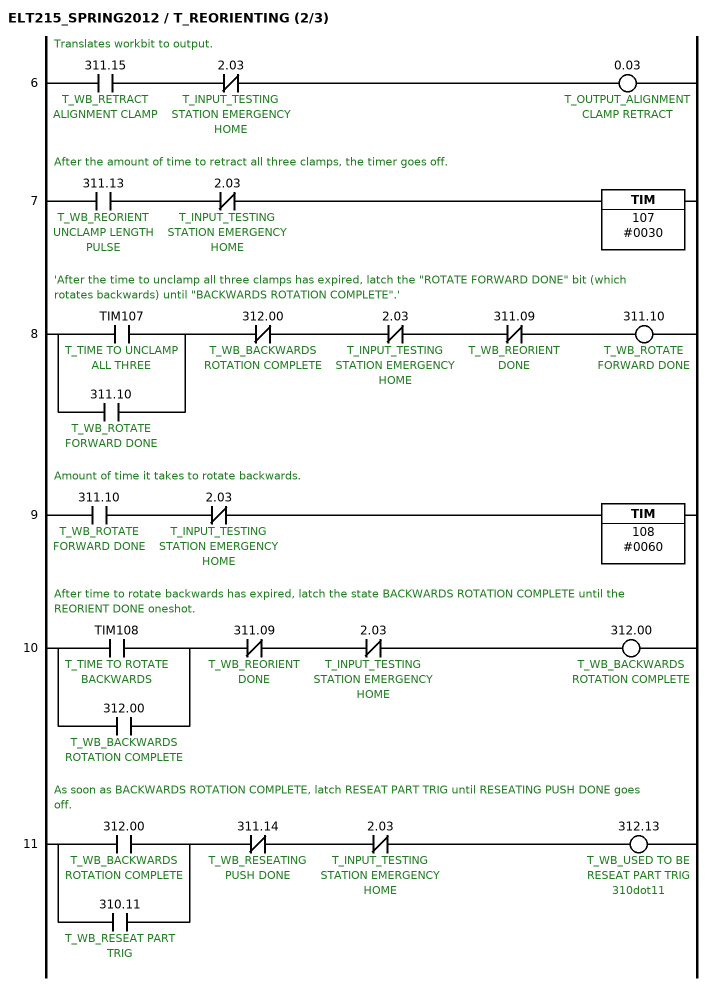
; [picture p24: ELT215_SPRING2012 / T_REORIENTING, rungs 6-11]
; rung 6: Translates workbit to output.
LD 311.15  ; T_WB_RETRACT ALIGNMENT CLAMP
ANDNOT 2.03  ; T_INPUT_TESTING STATION EMERGENCY HOME
OUT 0.03  ; T_OUTPUT_ALIGNMENT CLAMP RETRACT
; rung 7: After the amount of time to retract all three clamps, the timer goes off.
LD 311.13  ; T_WB_REORIENT UNCLAMP LENGTH PULSE
ANDNOT 2.03  ; T_INPUT_TESTING STATION EMERGENCY HOME
TIM 107 #0030
; rung 8: 'After the time to unclamp all three clamps has expired, latch the "ROTATE FORWARD DONE" bit (which rotates backwards) until "BACKWARDS ROTATION COMPLETE".'
LD TIM107  ; T_TIME TO UNCLAMP ALL THREE
OR 311.10  ; T_WB_ROTATE FORWARD DONE
ANDNOT 312.00  ; T_WB_BACKWARDS ROTATION COMPLETE
ANDNOT 2.03  ; T_INPUT_TESTING STATION EMERGENCY HOME
ANDNOT 311.09  ; T_WB_REORIENT DONE
OUT 311.10  ; T_WB_ROTATE FORWARD DONE
; rung 9: Amount of time it takes to rotate backwards.
LD 311.10  ; T_WB_ROTATE FORWARD DONE
ANDNOT 2.03  ; T_INPUT_TESTING STATION EMERGENCY HOME
TIM 108 #0060
; rung 10: After time to rotate backwards has expired, latch the state BACKWARDS ROTATION COMPLETE until the REORIENT DONE oneshot.
LD TIM108  ; T_TIME TO ROTATE BACKWARDS
OR 312.00  ; T_WB_BACKWARDS ROTATION COMPLETE
ANDNOT 311.09  ; T_WB_REORIENT DONE
ANDNOT 2.03  ; T_INPUT_TESTING STATION EMERGENCY HOME
OUT 312.00  ; T_WB_BACKWARDS ROTATION COMPLETE
; rung 11: As soon as BACKWARDS ROTATION COMPLETE, latch RESEAT PART TRIG until RESEATING PUSH DONE goes off.
LD 312.00  ; T_WB_BACKWARDS ROTATION COMPLETE
OR 310.11  ; T_WB_RESEAT PART TRIG
ANDNOT 311.14  ; T_WB_RESEATING PUSH DONE
ANDNOT 2.03  ; T_INPUT_TESTING STATION EMERGENCY HOME
OUT 312.13  ; T_WB_USED TO BE RESEAT PART TRIG 310dot11

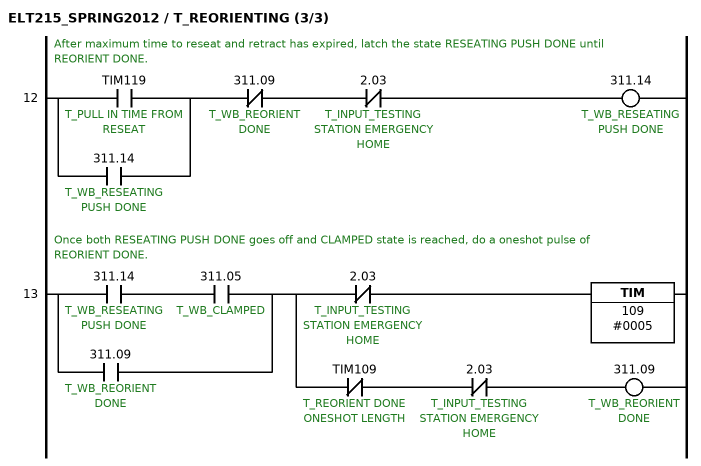
; rung 12: After maximum time to reseat and retract has expired, latch the state RESEATING PUSH DONE until REORIENT DONE.
LD TIM119  ; T_PULL IN TIME FROM RESEAT
OR 311.14  ; T_WB_RESEATING PUSH DONE
ANDNOT 311.09  ; T_WB_REORIENT DONE
ANDNOT 2.03  ; T_INPUT_TESTING STATION EMERGENCY HOME
OUT 311.14  ; T_WB_RESEATING PUSH DONE
; rung 13: Once both RESEATING PUSH DONE goes off and CLAMPED state is reached, do a oneshot pulse of REORIENT DONE.
LD 311.14  ; T_WB_RESEATING PUSH DONE
AND 311.05  ; T_WB_CLAMPED
OR 311.09  ; T_WB_REORIENT DONE
OUT TR0
ANDNOT 2.03  ; T_INPUT_TESTING STATION EMERGENCY HOME
TIM 109 #0005
LD TR0
ANDNOT TIM109  ; T_REORIENT DONE ONESHOT LENGTH
ANDNOT 2.03  ; T_INPUT_TESTING STATION EMERGENCY HOME
OUT 311.09  ; T_WB_REORIENT DONE

### Section T_HOLD_FOR_TESTING
; Ladder logic that can accept a tier 2 request to hold the part for testing (identified as being properly oriented) and can perform the actions to hold the piece, run the test sequence, and then eject the piece from the system.

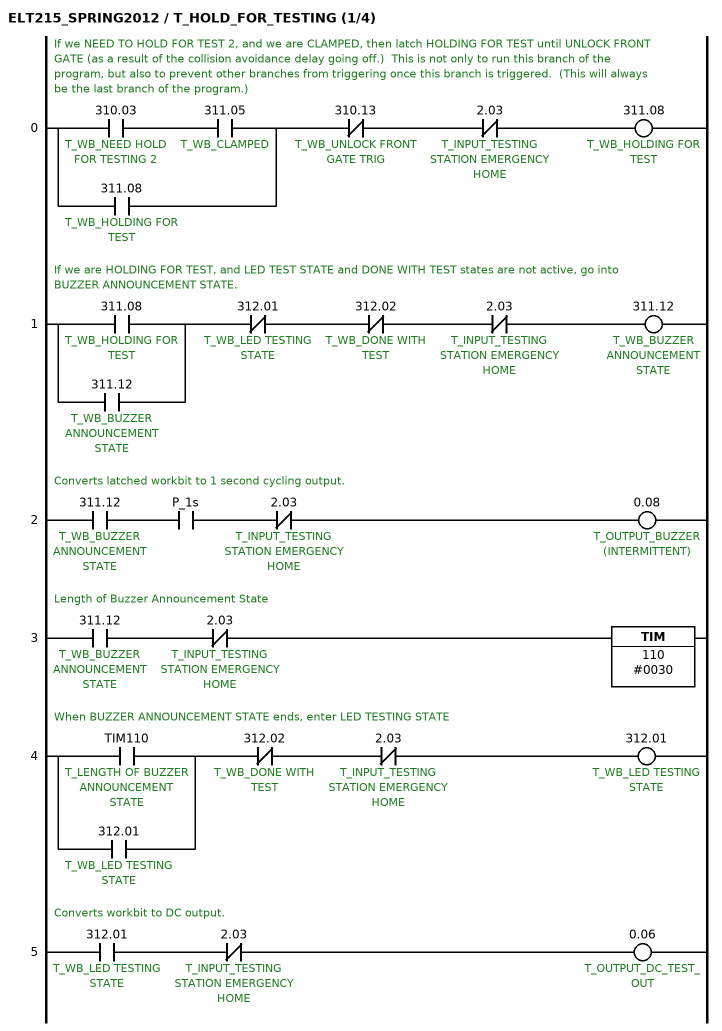
; rung 0: If we NEED TO HOLD FOR TEST 2, and we are CLAMPED, then latch HOLDING FOR TEST until UNLOCK FRONT GATE (as a result of the collision avoidance delay going off.)  This is not only to run this branch of the program, but also to prevent other branches from triggering once this branch is triggered.  (This will always be the last branch of the program.)
LD 310.03  ; T_WB_NEED HOLD FOR TESTING 2
AND 311.05  ; T_WB_CLAMPED
OR 311.08  ; T_WB_HOLDING FOR TEST
ANDNOT 310.13  ; T_WB_UNLOCK FRONT GATE TRIG
ANDNOT 2.03  ; T_INPUT_TESTING STATION EMERGENCY HOME
OUT 311.08  ; T_WB_HOLDING FOR TEST
; rung 1: If we are HOLDING FOR TEST, and LED TEST STATE and DONE WITH TEST states are not active, go into BUZZER ANNOUNCEMENT STATE.
LD 311.08  ; T_WB_HOLDING FOR TEST
OR 311.12  ; T_WB_BUZZER ANNOUNCEMENT STATE
ANDNOT 312.01  ; T_WB_LED TESTING STATE
ANDNOT 312.02  ; T_WB_DONE WITH TEST
ANDNOT 2.03  ; T_INPUT_TESTING STATION EMERGENCY HOME
OUT 311.12  ; T_WB_BUZZER ANNOUNCEMENT STATE
; rung 2: Converts latched workbit to 1 second cycling output.
LD 311.12  ; T_WB_BUZZER ANNOUNCEMENT STATE
AND P_1s
ANDNOT 2.03  ; T_INPUT_TESTING STATION EMERGENCY HOME
OUT 0.08  ; T_OUTPUT_BUZZER (INTERMITTENT)
; rung 3: Length of Buzzer Announcement State
LD 311.12  ; T_WB_BUZZER ANNOUNCEMENT STATE
ANDNOT 2.03  ; T_INPUT_TESTING STATION EMERGENCY HOME
TIM 110 #0030
; rung 4: When BUZZER ANNOUNCEMENT STATE ends, enter LED TESTING STATE
LD TIM110  ; T_LENGTH OF BUZZER ANNOUNCEMENT STATE
OR 312.01  ; T_WB_LED TESTING STATE
ANDNOT 312.02  ; T_WB_DONE WITH TEST
ANDNOT 2.03  ; T_INPUT_TESTING STATION EMERGENCY HOME
OUT 312.01  ; T_WB_LED TESTING STATE
; rung 5: Converts workbit to DC output.
LD 312.01  ; T_WB_LED TESTING STATE
ANDNOT 2.03  ; T_INPUT_TESTING STATION EMERGENCY HOME
OUT 0.06  ; T_OUTPUT_DC_TEST_OUT

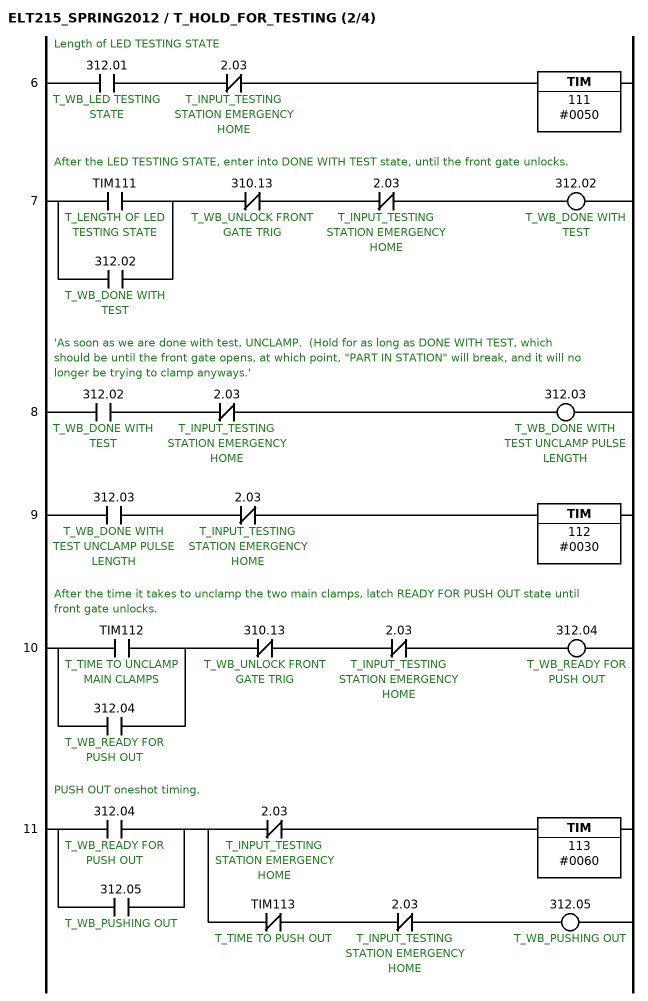
; rung 6: Length of LED TESTING STATE
LD 312.01  ; T_WB_LED TESTING STATE
ANDNOT 2.03  ; T_INPUT_TESTING STATION EMERGENCY HOME
TIM 111 #0050
; rung 7: After the LED TESTING STATE, enter into DONE WITH TEST state, until the front gate unlocks.
LD TIM111  ; T_LENGTH OF LED TESTING STATE
OR 312.02  ; T_WB_DONE WITH TEST
ANDNOT 310.13  ; T_WB_UNLOCK FRONT GATE TRIG
ANDNOT 2.03  ; T_INPUT_TESTING STATION EMERGENCY HOME
OUT 312.02  ; T_WB_DONE WITH TEST
; rung 8: 'As soon as we are done with test, UNCLAMP.  (Hold for as long as DONE WITH TEST, which should be until the front gate opens, at which point, "PART IN STATION" will break, and it will no longer be trying to clamp anyways.'
LD 312.02  ; T_WB_DONE WITH TEST
ANDNOT 2.03  ; T_INPUT_TESTING STATION EMERGENCY HOME
OUT 312.03  ; T_WB_DONE WITH TEST UNCLAMP PULSE LENGTH
; rung 9
LD 312.03  ; T_WB_DONE WITH TEST UNCLAMP PULSE LENGTH
ANDNOT 2.03  ; T_INPUT_TESTING STATION EMERGENCY HOME
TIM 112 #0030
; rung 10: After the time it takes to unclamp the two main clamps, latch READY FOR PUSH OUT state until front gate unlocks.
LD TIM112  ; T_TIME TO UNCLAMP MAIN CLAMPS
OR 312.04  ; T_WB_READY FOR PUSH OUT
ANDNOT 310.13  ; T_WB_UNLOCK FRONT GATE TRIG
ANDNOT 2.03  ; T_INPUT_TESTING STATION EMERGENCY HOME
OUT 312.04  ; T_WB_READY FOR PUSH OUT
; rung 11: PUSH OUT oneshot timing.
LD 312.04  ; T_WB_READY FOR PUSH OUT
OR 312.05  ; T_WB_PUSHING OUT
OUT TR0
ANDNOT 2.03  ; T_INPUT_TESTING STATION EMERGENCY HOME
TIM 113 #0060
LD TR0
ANDNOT TIM113  ; T_TIME TO PUSH OUT
ANDNOT 2.03  ; T_INPUT_TESTING STATION EMERGENCY HOME
OUT 312.05  ; T_WB_PUSHING OUT

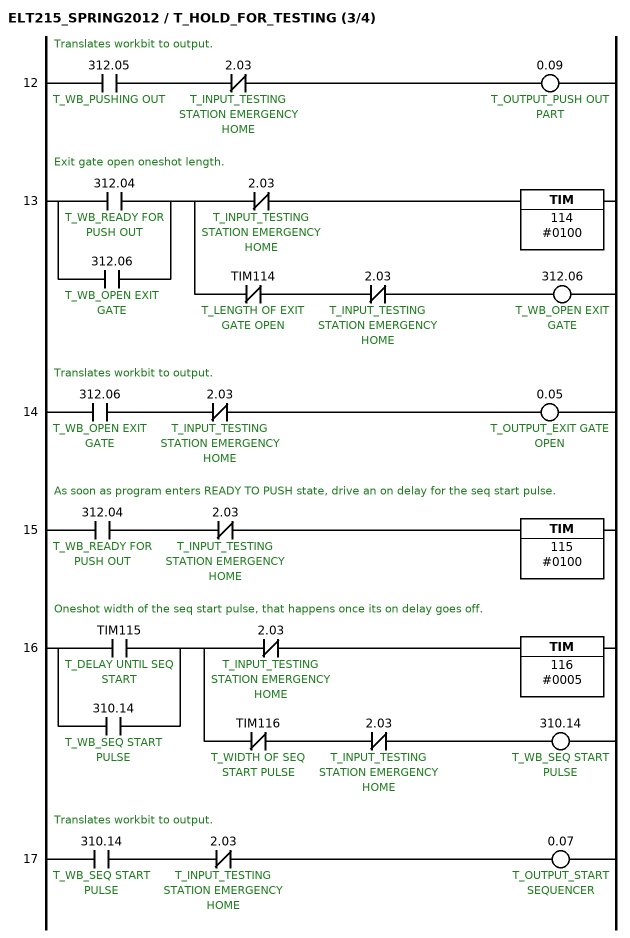
; rung 12: Translates workbit to output.
LD 312.05  ; T_WB_PUSHING OUT
ANDNOT 2.03  ; T_INPUT_TESTING STATION EMERGENCY HOME
OUT 0.09  ; T_OUTPUT_PUSH OUT PART
; rung 13: Exit gate open oneshot length.
LD 312.04  ; T_WB_READY FOR PUSH OUT
OR 312.06  ; T_WB_OPEN EXIT GATE
OUT TR0
ANDNOT 2.03  ; T_INPUT_TESTING STATION EMERGENCY HOME
TIM 114 #0100
LD TR0
ANDNOT TIM114  ; T_LENGTH OF EXIT GATE OPEN
ANDNOT 2.03  ; T_INPUT_TESTING STATION EMERGENCY HOME
OUT 312.06  ; T_WB_OPEN EXIT GATE
; rung 14: Translates workbit to output.
LD 312.06  ; T_WB_OPEN EXIT GATE
ANDNOT 2.03  ; T_INPUT_TESTING STATION EMERGENCY HOME
OUT 0.05  ; T_OUTPUT_EXIT GATE OPEN
; rung 15: As soon as program enters READY TO PUSH state, drive an on delay for the seq start pulse.
LD 312.04  ; T_WB_READY FOR PUSH OUT
ANDNOT 2.03  ; T_INPUT_TESTING STATION EMERGENCY HOME
TIM 115 #0100
; rung 16: Oneshot width of the seq start pulse, that happens once its on delay goes off.
LD TIM115  ; T_DELAY UNTIL SEQ START
OR 310.14  ; T_WB_SEQ START PULSE
OUT TR0
ANDNOT 2.03  ; T_INPUT_TESTING STATION EMERGENCY HOME
TIM 116 #0005
LD TR0
ANDNOT TIM116  ; T_WIDTH OF SEQ START PULSE
ANDNOT 2.03  ; T_INPUT_TESTING STATION EMERGENCY HOME
OUT 310.14  ; T_WB_SEQ START PULSE
; rung 17: Translates workbit to output.
LD 310.14  ; T_WB_SEQ START PULSE
ANDNOT 2.03  ; T_INPUT_TESTING STATION EMERGENCY HOME
OUT 0.07  ; T_OUTPUT_START SEQUENCER

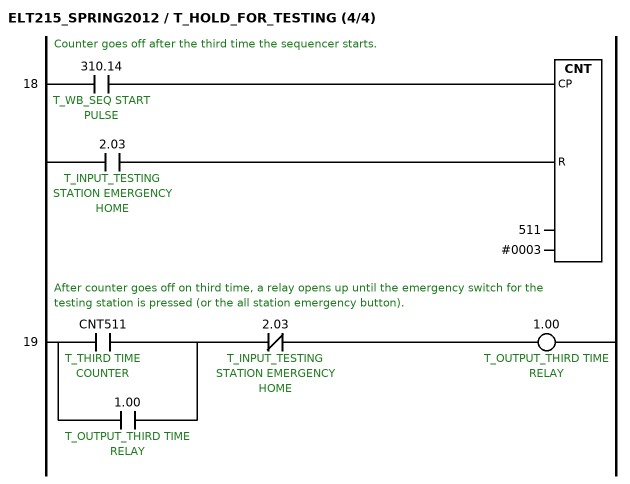
; rung 18: Counter goes off after the third time the sequencer starts.
LD 310.14  ; T_WB_SEQ START PULSE
LD 2.03  ; T_INPUT_TESTING STATION EMERGENCY HOME
CNT 511 #0003
; rung 19: After counter goes off on third time, a relay opens up until the emergency switch for the testing station is pressed (or the all station emergency button).
LD CNT511  ; T_THIRD TIME COUNTER
OR 1.00  ; T_OUTPUT_THIRD TIME RELAY
ANDNOT 2.03  ; T_INPUT_TESTING STATION EMERGENCY HOME
OUT 1.00  ; T_OUTPUT_THIRD TIME RELAY

### Section T_SYSTEM_RESET_AND_ABORT
; Ladder logic that defines the two different ways the program can end and reset.  A. Through an abort command  B. Through a SEQ START pulse, which will then get delayed to avoid a possible collision if the next part comes in properly oriented.

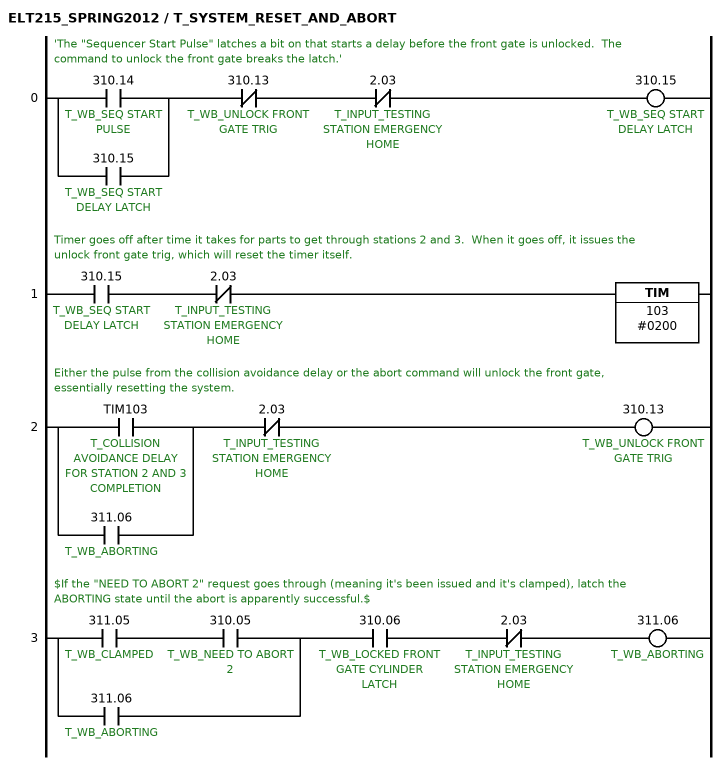
; rung 0: 'The "Sequencer Start Pulse" latches a bit on that starts a delay before the front gate is unlocked.  The command to unlock the front gate breaks the latch.'
LD 310.14  ; T_WB_SEQ START PULSE
OR 310.15  ; T_WB_SEQ START DELAY LATCH
ANDNOT 310.13  ; T_WB_UNLOCK FRONT GATE TRIG
ANDNOT 2.03  ; T_INPUT_TESTING STATION EMERGENCY HOME
OUT 310.15  ; T_WB_SEQ START DELAY LATCH
; rung 1: Timer goes off after time it takes for parts to get through stations 2 and 3.  When it goes off, it issues the unlock front gate trig, which will reset the timer itself.
LD 310.15  ; T_WB_SEQ START DELAY LATCH
ANDNOT 2.03  ; T_INPUT_TESTING STATION EMERGENCY HOME
TIM 103 #0200
; rung 2: Either the pulse from the collision avoidance delay or the abort command will unlock the front gate, essentially resetting the system.
LD TIM103  ; T_COLLISION AVOIDANCE DELAY FOR STATION 2 AND 3 COMPLETION
OR 311.06  ; T_WB_ABORTING
ANDNOT 2.03  ; T_INPUT_TESTING STATION EMERGENCY HOME
OUT 310.13  ; T_WB_UNLOCK FRONT GATE TRIG
; rung 3: $If the "NEED TO ABORT 2" request goes through (meaning it's been issued and it's clamped), latch the ABORTING state until the abort is apparently successful.$
LD 311.05  ; T_WB_CLAMPED
AND 310.05  ; T_WB_NEED TO ABORT 2
OR 311.06  ; T_WB_ABORTING
AND 310.06  ; T_WB_LOCKED FRONT GATE CYLINDER LATCH
ANDNOT 2.03  ; T_INPUT_TESTING STATION EMERGENCY HOME
OUT 311.06  ; T_WB_ABORTING

### Section T_OBSERVATION_ONLY

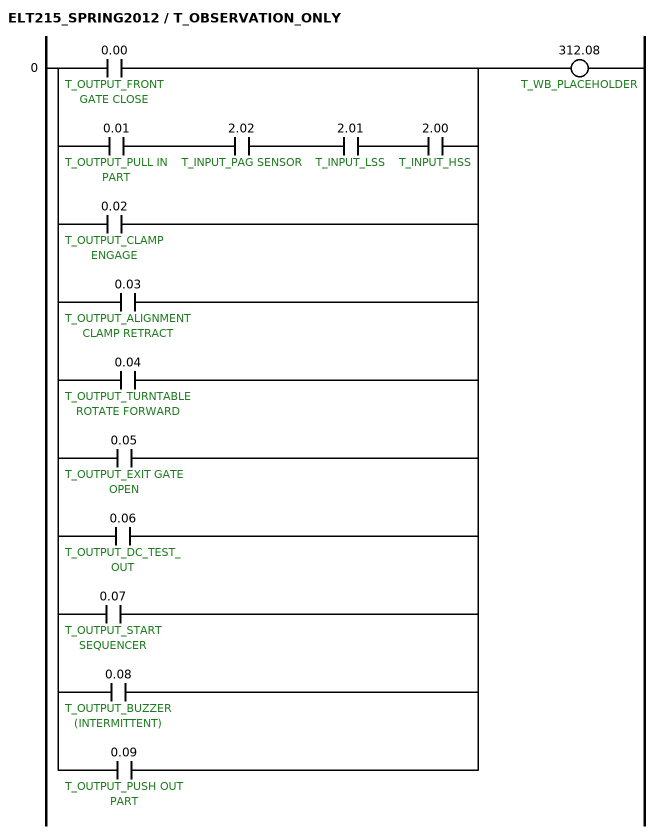
; rung 0
LD 0.00  ; T_OUTPUT_FRONT GATE CLOSE
LD 0.01  ; T_OUTPUT_PULL IN PART
AND 2.02  ; T_INPUT_PAG SENSOR
AND 2.01  ; T_INPUT_LSS
AND 2.00  ; T_INPUT_HSS
ORLD
LD 0.02  ; T_OUTPUT_CLAMP ENGAGE
OR 0.03  ; T_OUTPUT_ALIGNMENT CLAMP RETRACT
OR 0.04  ; T_OUTPUT_TURNTABLE ROTATE FORWARD
OR 0.05  ; T_OUTPUT_EXIT GATE OPEN
OR 0.06  ; T_OUTPUT_DC_TEST_OUT
OR 0.07  ; T_OUTPUT_START SEQUENCER
OR 0.08  ; T_OUTPUT_BUZZER (INTERMITTENT)
OR 0.09  ; T_OUTPUT_PUSH OUT PART
ORLD
OUT 312.08  ; T_WB_PLACEHOLDER

### Section F_FEEDER_SEQUENCE_TIME
; 'Offset from T=0, contains timings for the ejection of each part, as well as the "SEQUENCE OVER" point.  For example, if parts are supposed to come out at ten second intervals, part 1 would be released at 0, part 2 at 10, part 3 at 20, etc.'

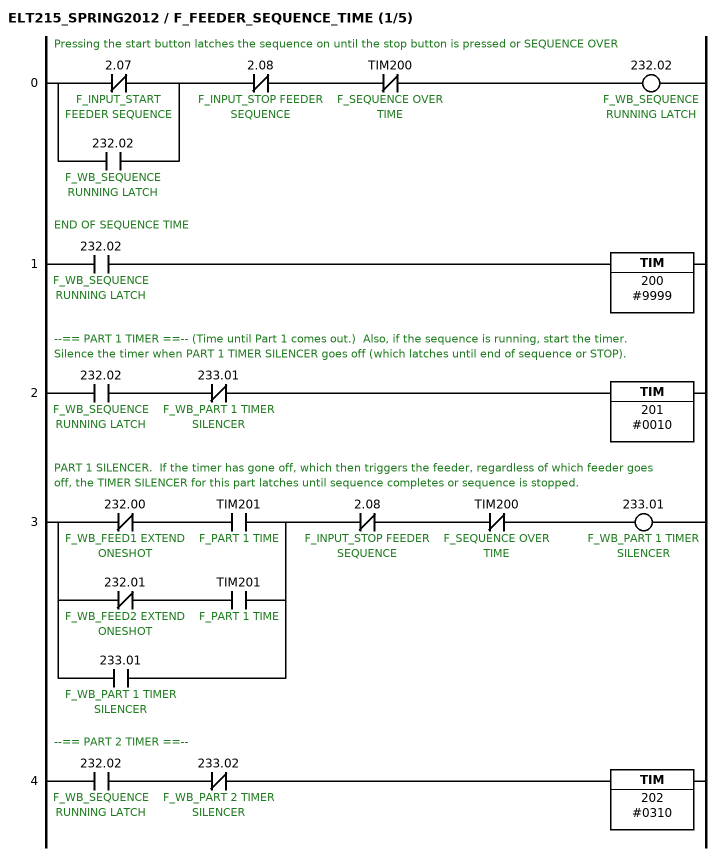
; rung 0: Pressing the start button latches the sequence on until the stop button is pressed or SEQUENCE OVER
LDNOT 2.07  ; F_INPUT_START FEEDER SEQUENCE
OR 232.02  ; F_WB_SEQUENCE RUNNING LATCH
ANDNOT 2.08  ; F_INPUT_STOP FEEDER SEQUENCE
ANDNOT TIM200  ; F_SEQUENCE OVER TIME
OUT 232.02  ; F_WB_SEQUENCE RUNNING LATCH
; rung 1: END OF SEQUENCE TIME
LD 232.02  ; F_WB_SEQUENCE RUNNING LATCH
TIM 200 #9999
; rung 2: --== PART 1 TIMER ==-- (Time until Part 1 comes out.)  Also, if the sequence is running, start the timer.  Silence the timer when PART 1 TIMER SILENCER goes off (which latches until end of sequence or STOP).
LD 232.02  ; F_WB_SEQUENCE RUNNING LATCH
ANDNOT 233.01  ; F_WB_PART 1 TIMER SILENCER
TIM 201 #0010
; rung 3: PART 1 SILENCER.  If the timer has gone off, which then triggers the feeder, regardless of which feeder goes off, the TIMER SILENCER for this part latches until sequence completes or sequence is stopped.
LDNOT 232.00  ; F_WB_FEED1 EXTEND ONESHOT
AND TIM201  ; F_PART 1 TIME
LDNOT 232.01  ; F_WB_FEED2 EXTEND ONESHOT
AND TIM201  ; F_PART 1 TIME
ORLD
OR 233.01  ; F_WB_PART 1 TIMER SILENCER
ANDNOT 2.08  ; F_INPUT_STOP FEEDER SEQUENCE
ANDNOT TIM200  ; F_SEQUENCE OVER TIME
OUT 233.01  ; F_WB_PART 1 TIMER SILENCER
; rung 4: --== PART 2 TIMER ==--
LD 232.02  ; F_WB_SEQUENCE RUNNING LATCH
ANDNOT 233.02  ; F_WB_PART 2 TIMER SILENCER
TIM 202 #0310

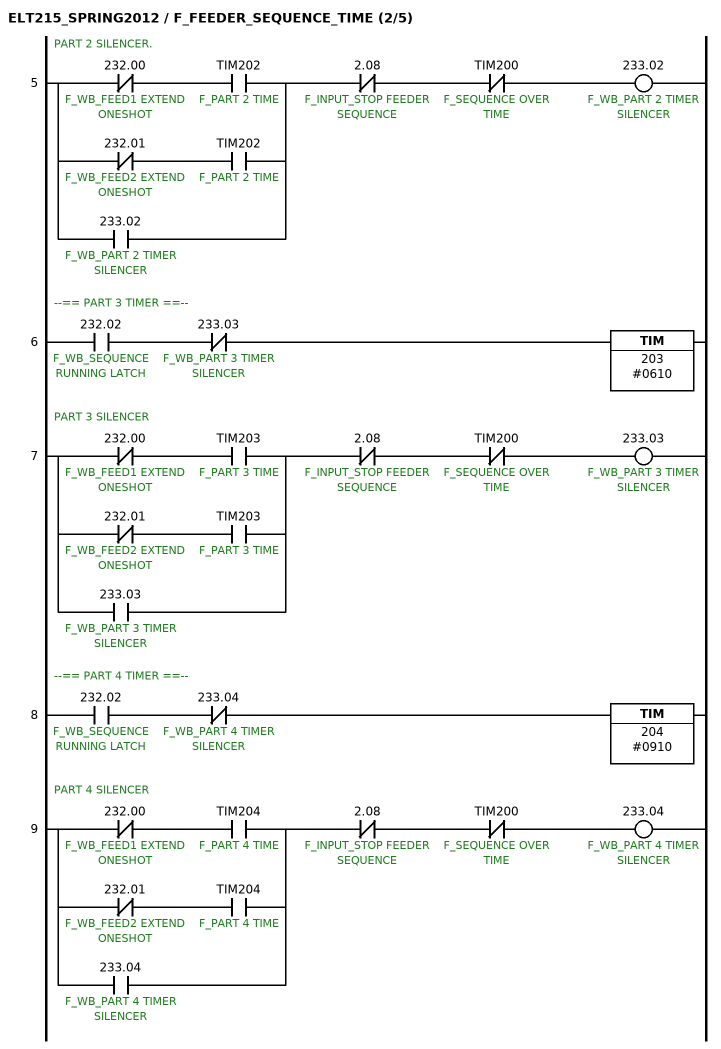
; rung 5: PART 2 SILENCER.
LDNOT 232.00  ; F_WB_FEED1 EXTEND ONESHOT
AND TIM202  ; F_PART 2 TIME
LDNOT 232.01  ; F_WB_FEED2 EXTEND ONESHOT
AND TIM202  ; F_PART 2 TIME
ORLD
OR 233.02  ; F_WB_PART 2 TIMER SILENCER
ANDNOT 2.08  ; F_INPUT_STOP FEEDER SEQUENCE
ANDNOT TIM200  ; F_SEQUENCE OVER TIME
OUT 233.02  ; F_WB_PART 2 TIMER SILENCER
; rung 6: --== PART 3 TIMER ==--
LD 232.02  ; F_WB_SEQUENCE RUNNING LATCH
ANDNOT 233.03  ; F_WB_PART 3 TIMER SILENCER
TIM 203 #0610
; rung 7: PART 3 SILENCER
LDNOT 232.00  ; F_WB_FEED1 EXTEND ONESHOT
AND TIM203  ; F_PART 3 TIME
LDNOT 232.01  ; F_WB_FEED2 EXTEND ONESHOT
AND TIM203  ; F_PART 3 TIME
ORLD
OR 233.03  ; F_WB_PART 3 TIMER SILENCER
ANDNOT 2.08  ; F_INPUT_STOP FEEDER SEQUENCE
ANDNOT TIM200  ; F_SEQUENCE OVER TIME
OUT 233.03  ; F_WB_PART 3 TIMER SILENCER
; rung 8: --== PART 4 TIMER ==--
LD 232.02  ; F_WB_SEQUENCE RUNNING LATCH
ANDNOT 233.04  ; F_WB_PART 4 TIMER SILENCER
TIM 204 #0910
; rung 9: PART 4 SILENCER
LDNOT 232.00  ; F_WB_FEED1 EXTEND ONESHOT
AND TIM204  ; F_PART 4 TIME
LDNOT 232.01  ; F_WB_FEED2 EXTEND ONESHOT
AND TIM204  ; F_PART 4 TIME
ORLD
OR 233.04  ; F_WB_PART 4 TIMER SILENCER
ANDNOT 2.08  ; F_INPUT_STOP FEEDER SEQUENCE
ANDNOT TIM200  ; F_SEQUENCE OVER TIME
OUT 233.04  ; F_WB_PART 4 TIMER SILENCER

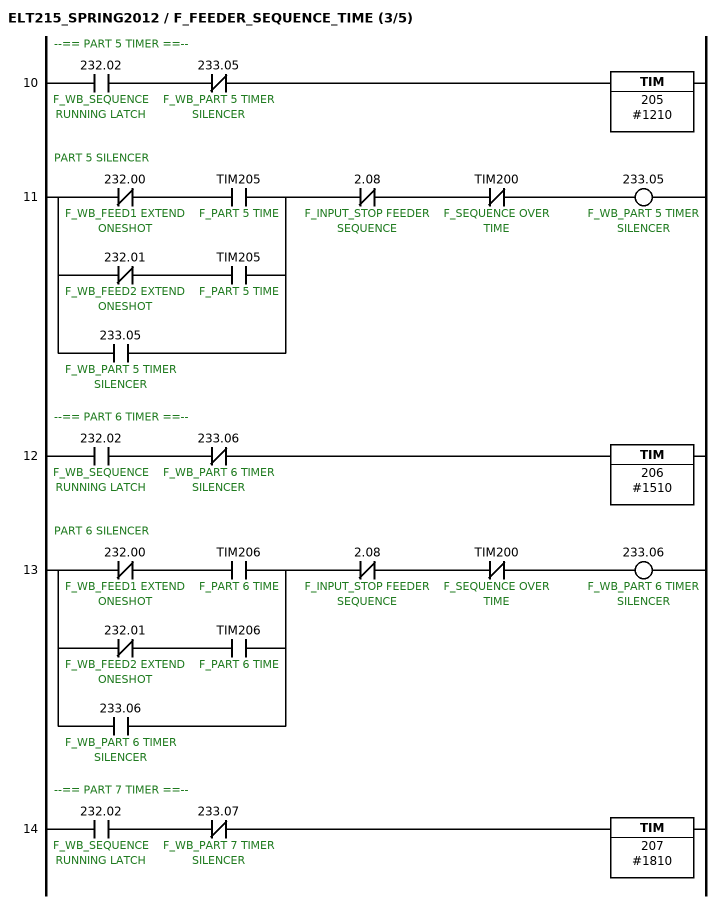
; rung 10: --== PART 5 TIMER ==--
LD 232.02  ; F_WB_SEQUENCE RUNNING LATCH
ANDNOT 233.05  ; F_WB_PART 5 TIMER SILENCER
TIM 205 #1210
; rung 11: PART 5 SILENCER
LDNOT 232.00  ; F_WB_FEED1 EXTEND ONESHOT
AND TIM205  ; F_PART 5 TIME
LDNOT 232.01  ; F_WB_FEED2 EXTEND ONESHOT
AND TIM205  ; F_PART 5 TIME
ORLD
OR 233.05  ; F_WB_PART 5 TIMER SILENCER
ANDNOT 2.08  ; F_INPUT_STOP FEEDER SEQUENCE
ANDNOT TIM200  ; F_SEQUENCE OVER TIME
OUT 233.05  ; F_WB_PART 5 TIMER SILENCER
; rung 12: --== PART 6 TIMER ==--
LD 232.02  ; F_WB_SEQUENCE RUNNING LATCH
ANDNOT 233.06  ; F_WB_PART 6 TIMER SILENCER
TIM 206 #1510
; rung 13: PART 6 SILENCER
LDNOT 232.00  ; F_WB_FEED1 EXTEND ONESHOT
AND TIM206  ; F_PART 6 TIME
LDNOT 232.01  ; F_WB_FEED2 EXTEND ONESHOT
AND TIM206  ; F_PART 6 TIME
ORLD
OR 233.06  ; F_WB_PART 6 TIMER SILENCER
ANDNOT 2.08  ; F_INPUT_STOP FEEDER SEQUENCE
ANDNOT TIM200  ; F_SEQUENCE OVER TIME
OUT 233.06  ; F_WB_PART 6 TIMER SILENCER
; rung 14: --== PART 7 TIMER ==--
LD 232.02  ; F_WB_SEQUENCE RUNNING LATCH
ANDNOT 233.07  ; F_WB_PART 7 TIMER SILENCER
TIM 207 #1810

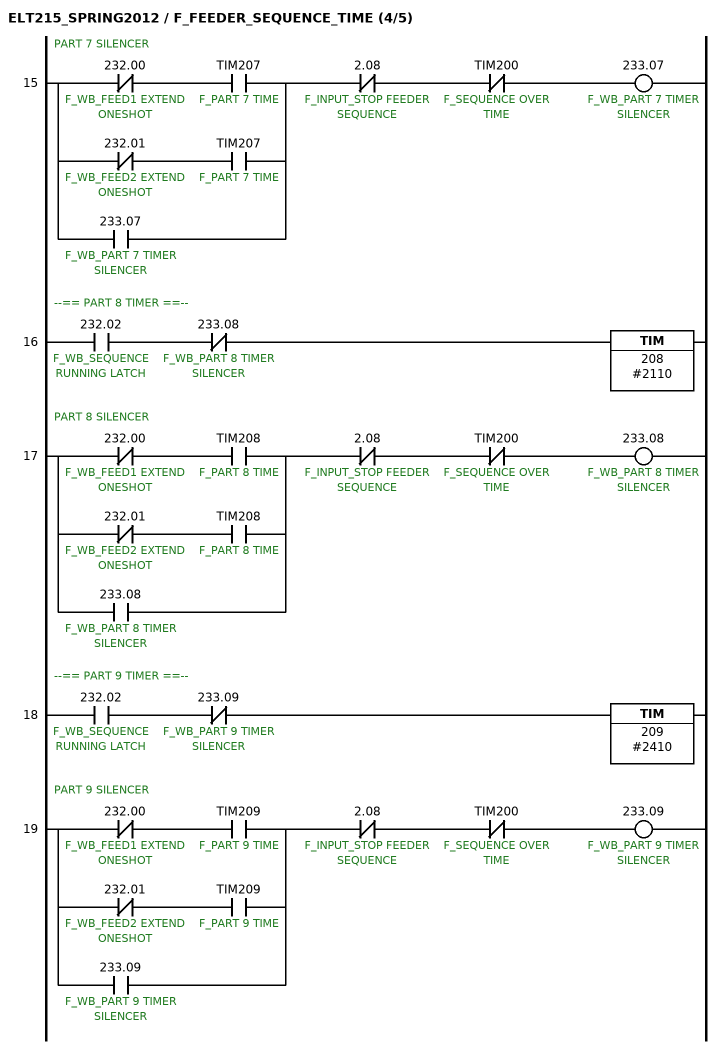
; rung 15: PART 7 SILENCER
LDNOT 232.00  ; F_WB_FEED1 EXTEND ONESHOT
AND TIM207  ; F_PART 7 TIME
LDNOT 232.01  ; F_WB_FEED2 EXTEND ONESHOT
AND TIM207  ; F_PART 7 TIME
ORLD
OR 233.07  ; F_WB_PART 7 TIMER SILENCER
ANDNOT 2.08  ; F_INPUT_STOP FEEDER SEQUENCE
ANDNOT TIM200  ; F_SEQUENCE OVER TIME
OUT 233.07  ; F_WB_PART 7 TIMER SILENCER
; rung 16: --== PART 8 TIMER ==--
LD 232.02  ; F_WB_SEQUENCE RUNNING LATCH
ANDNOT 233.08  ; F_WB_PART 8 TIMER SILENCER
TIM 208 #2110
; rung 17: PART 8 SILENCER
LDNOT 232.00  ; F_WB_FEED1 EXTEND ONESHOT
AND TIM208  ; F_PART 8 TIME
LDNOT 232.01  ; F_WB_FEED2 EXTEND ONESHOT
AND TIM208  ; F_PART 8 TIME
ORLD
OR 233.08  ; F_WB_PART 8 TIMER SILENCER
ANDNOT 2.08  ; F_INPUT_STOP FEEDER SEQUENCE
ANDNOT TIM200  ; F_SEQUENCE OVER TIME
OUT 233.08  ; F_WB_PART 8 TIMER SILENCER
; rung 18: --== PART 9 TIMER ==--
LD 232.02  ; F_WB_SEQUENCE RUNNING LATCH
ANDNOT 233.09  ; F_WB_PART 9 TIMER SILENCER
TIM 209 #2410
; rung 19: PART 9 SILENCER
LDNOT 232.00  ; F_WB_FEED1 EXTEND ONESHOT
AND TIM209  ; F_PART 9 TIME
LDNOT 232.01  ; F_WB_FEED2 EXTEND ONESHOT
AND TIM209  ; F_PART 9 TIME
ORLD
OR 233.09  ; F_WB_PART 9 TIMER SILENCER
ANDNOT 2.08  ; F_INPUT_STOP FEEDER SEQUENCE
ANDNOT TIM200  ; F_SEQUENCE OVER TIME
OUT 233.09  ; F_WB_PART 9 TIMER SILENCER

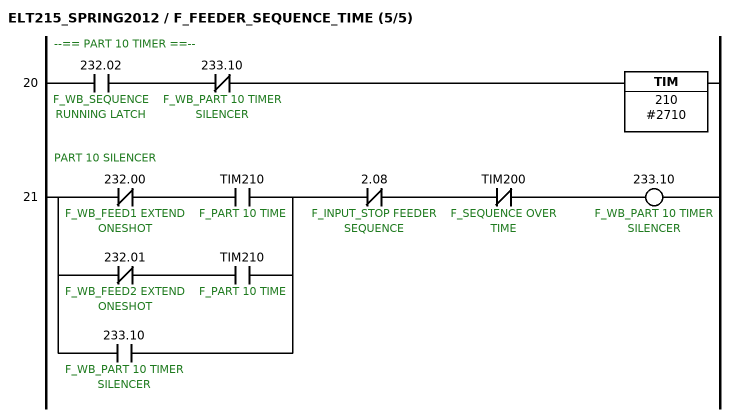
; rung 20: --== PART 10 TIMER ==--
LD 232.02  ; F_WB_SEQUENCE RUNNING LATCH
ANDNOT 233.10  ; F_WB_PART 10 TIMER SILENCER
TIM 210 #2710
; rung 21: PART 10 SILENCER
LDNOT 232.00  ; F_WB_FEED1 EXTEND ONESHOT
AND TIM210  ; F_PART 10 TIME
LDNOT 232.01  ; F_WB_FEED2 EXTEND ONESHOT
AND TIM210  ; F_PART 10 TIME
ORLD
OR 233.10  ; F_WB_PART 10 TIMER SILENCER
ANDNOT 2.08  ; F_INPUT_STOP FEEDER SEQUENCE
ANDNOT TIM200  ; F_SEQUENCE OVER TIME
OUT 233.10  ; F_WB_PART 10 TIMER SILENCER

### Section F_FEEDER_SEQUENCE_ORDER
; When the timer for a specific part goes off, that signal is sent to either Feeder 1 or Feeder 2.  These first two rungs determine which go where.

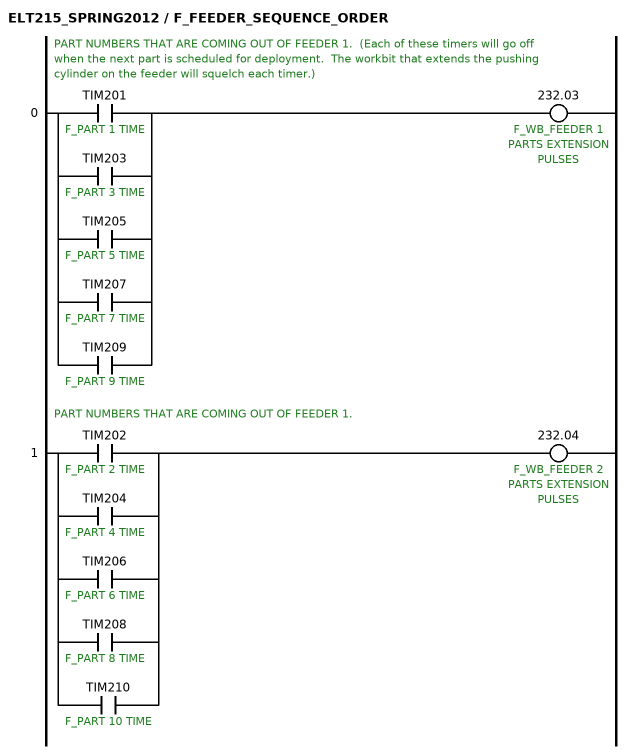
; rung 0: PART NUMBERS THAT ARE COMING OUT OF FEEDER 1.  (Each of these timers will go off when the next part is scheduled for deployment.  The workbit that extends the pushing cylinder on the feeder will squelch each timer.)
LD TIM201  ; F_PART 1 TIME
OR TIM203  ; F_PART 3 TIME
OR TIM205  ; F_PART 5 TIME
OR TIM207  ; F_PART 7 TIME
OR TIM209  ; F_PART 9 TIME
OUT 232.03  ; F_WB_FEEDER 1 PARTS EXTENSION PULSES
; rung 1: PART NUMBERS THAT ARE COMING OUT OF FEEDER 1.
LD TIM202  ; F_PART 2 TIME
OR TIM204  ; F_PART 4 TIME
OR TIM206  ; F_PART 6 TIME
OR TIM208  ; F_PART 8 TIME
OR TIM210  ; F_PART 10 TIME
OUT 232.04  ; F_WB_FEEDER 2 PARTS EXTENSION PULSES

### Section F_FEEDER_PUSH_TIMING
; Contains the oneshot durations for the cylinder of Feeder 1 and the cylinder for Feeder 2.

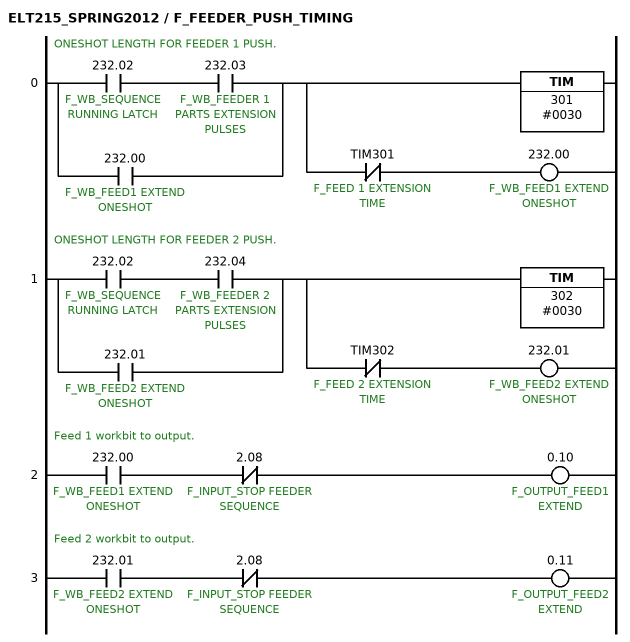
; rung 0: ONESHOT LENGTH FOR FEEDER 1 PUSH.
LD 232.02  ; F_WB_SEQUENCE RUNNING LATCH
AND 232.03  ; F_WB_FEEDER 1 PARTS EXTENSION PULSES
OR 232.00  ; F_WB_FEED1 EXTEND ONESHOT
TIM 301 #0030
ANDNOT TIM301  ; F_FEED 1 EXTENSION TIME
OUT 232.00  ; F_WB_FEED1 EXTEND ONESHOT
; rung 1: ONESHOT LENGTH FOR FEEDER 2 PUSH.
LD 232.02  ; F_WB_SEQUENCE RUNNING LATCH
AND 232.04  ; F_WB_FEEDER 2 PARTS EXTENSION PULSES
OR 232.01  ; F_WB_FEED2 EXTEND ONESHOT
TIM 302 #0030
ANDNOT TIM302  ; F_FEED 2 EXTENSION TIME
OUT 232.01  ; F_WB_FEED2 EXTEND ONESHOT
; rung 2: Feed 1 workbit to output.
LD 232.00  ; F_WB_FEED1 EXTEND ONESHOT
ANDNOT 2.08  ; F_INPUT_STOP FEEDER SEQUENCE
OUT 0.10  ; F_OUTPUT_FEED1 EXTEND
; rung 3: Feed 2 workbit to output.
LD 232.01  ; F_WB_FEED2 EXTEND ONESHOT
ANDNOT 2.08  ; F_INPUT_STOP FEEDER SEQUENCE
OUT 0.11  ; F_OUTPUT_FEED2 EXTEND

### Section END
; rung 0
END(01)